TYPE AX5000_S_0384 :
STRUCT
	Amplifier_temperature:UINT;
END_STRUCT
END_TYPE

(* stored: Version 1.1.0.1, ProductVersion 3.1.4024.3
   DUT AX5000_S_0384: Id {f70ae038-74c6-4b8d-844e-14023dcd1624} *)
